// TIA Portal V17 export
// export: Created 2022-04-06T07:28:38.3800124Z, ExportSetting WithDefaults, DisplayName Totally Integrated Automation Portal, DisplayVersion V17, DisplayName TIA Portal Openness, DisplayVersion V17, DisplayName TIA Portal Version Control Interface, DisplayVersion V17, DisplayName TIA Portal Test Suite Advanced, DisplayVersion V17, DisplayName SINAMICS Startdrive Advanced, DisplayVersion V17, DisplayName SINAMICS Startdrive G130, G150, S120, S150, SINAMICS MV, S210, DisplayVersion V17, DisplayName SINAMICS Startdrive G110M, G120, G120C, G120D, G120P, G115D, DisplayVersion V17, DisplayName STEP 7 Professional, DisplayVersion V17, DisplayName STEP 7 Safety, DisplayVersion V17, DisplayName WinCC Advanced / Unified PC, DisplayVersion V17
FUNCTION_BLOCK "Motion"   // FB2, FBD
{ S7_Optimized_Access := 'TRUE' }
VERSION : 0.1
// stored: AutoNumber true, IsIECCheckEnabled true, IsRetainMemResEnabled false, MemoryReserve 100, SetENOAutomatically false, UDAEnableTagReadback false
   VAR
      MC_POWER_Instance { S7_SetPoint := 'True'} : MC_POWER;
      MC_RESET_Instance { S7_SetPoint := 'True'} : MC_RESET;
      MC_HOME_Instance { S7_SetPoint := 'True'} : MC_HOME;
      MC_MOVEVELOCITY_Instance { S7_SetPoint := 'True'} : MC_MOVEVELOCITY;
      MC_HALT_Instance { S7_SetPoint := 'True'} : MC_HALT;
      MC_POWER_Instance_1 { S7_SetPoint := 'True'} : MC_POWER;
      MC_RESET_Instance_1 { S7_SetPoint := 'True'} : MC_RESET;
      MC_HOME_Instance_1 { S7_SetPoint := 'True'} : MC_HOME;
      MC_MOVEVELOCITY_Instance_1 { S7_SetPoint := 'True'} : MC_MOVEVELOCITY;
      MC_HALT_Instance_1 { S7_SetPoint := 'True'} : MC_HALT;
      instMC_MOVEVELOCITY_SlsActive { S7_SetPoint := 'True'} : MC_MOVEVELOCITY;
      statSlsPtrig { S7_SetPoint := 'True'} : Bool;
   END_VAR
   VAR_TEMP   // added for the SCL form of the ladder/FBD networks
      _w1 : Bool;
   END_VAR
BEGIN

REGION Network 1
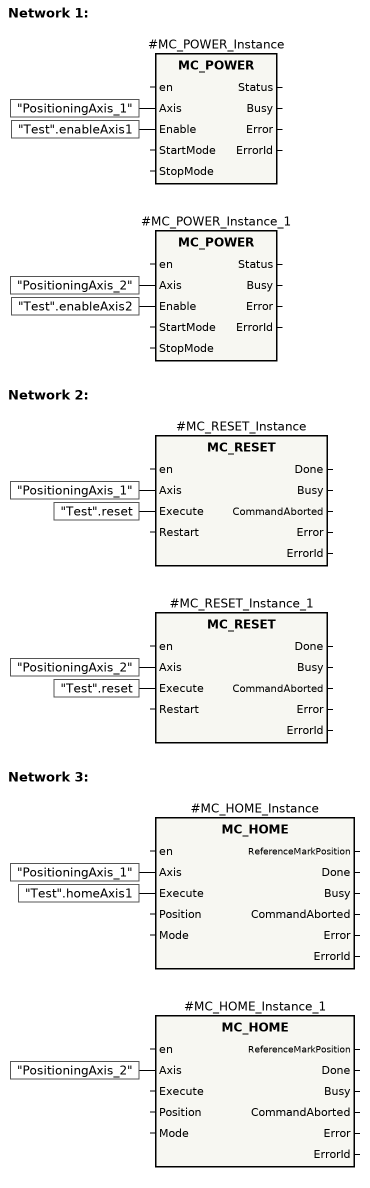
   #MC_POWER_Instance(Axis := "PositioningAxis_1", Enable := "Test".enableAxis1);   // MC_POWER
   #MC_POWER_Instance_1(Axis := "PositioningAxis_2", Enable := "Test".enableAxis2);   // MC_POWER
END_REGION

REGION Network 2
   #MC_RESET_Instance(Axis := "PositioningAxis_1", Execute := "Test".reset);   // MC_RESET
   #MC_RESET_Instance_1(Axis := "PositioningAxis_2", Execute := "Test".reset);   // MC_RESET
END_REGION

REGION Network 3
   #MC_HOME_Instance(Axis := "PositioningAxis_1", Execute := "Test".homeAxis1);   // MC_HOME
   #MC_HOME_Instance_1(Axis := "PositioningAxis_2");   // MC_HOME
END_REGION

REGION Network 4
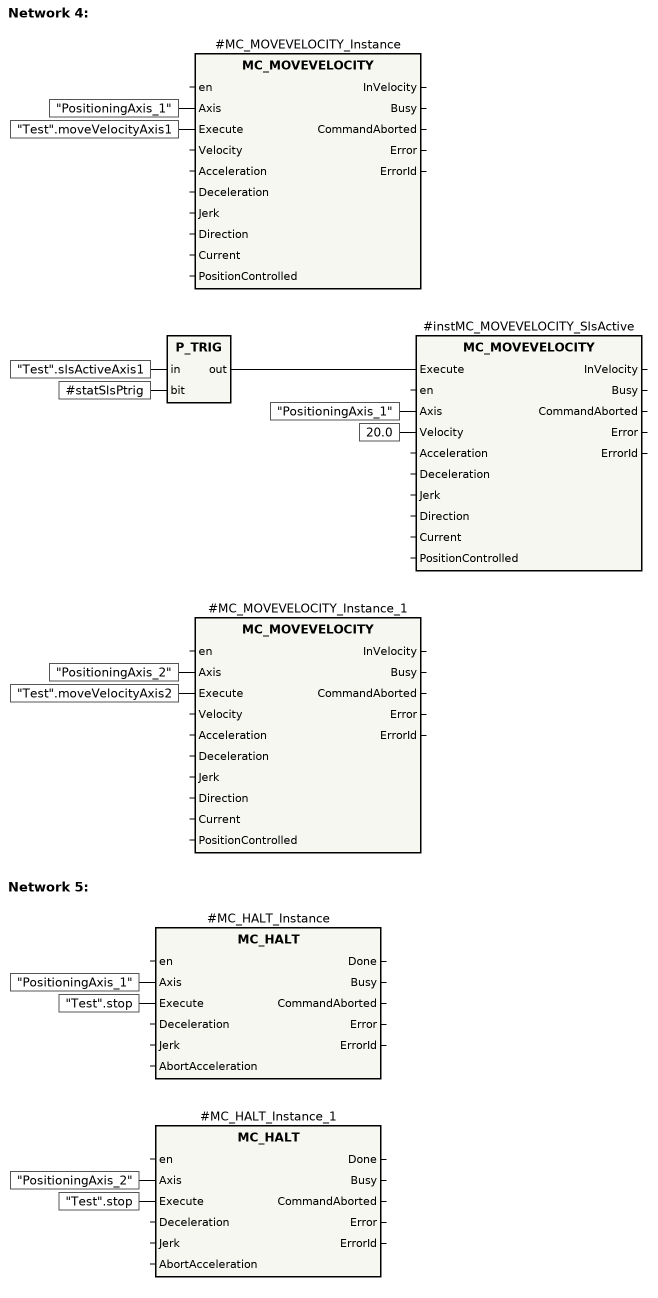
   #MC_MOVEVELOCITY_Instance(Axis := "PositioningAxis_1", Execute := "Test".moveVelocityAxis1);   // MC_MOVEVELOCITY
   #_w1 := "Test".slsActiveAxis1 AND NOT #statSlsPtrig;   // rising edge
   #statSlsPtrig := "Test".slsActiveAxis1;
   #instMC_MOVEVELOCITY_SlsActive(Execute := #_w1, Axis := "PositioningAxis_1", Velocity := 20.0);   // MC_MOVEVELOCITY
   #MC_MOVEVELOCITY_Instance_1(Axis := "PositioningAxis_2", Execute := "Test".moveVelocityAxis2);   // MC_MOVEVELOCITY
END_REGION

REGION Network 5
   #MC_HALT_Instance(Axis := "PositioningAxis_1", Execute := "Test".stop);   // MC_HALT
   #MC_HALT_Instance_1(Axis := "PositioningAxis_2", Execute := "Test".stop);   // MC_HALT
END_REGION
END_FUNCTION_BLOCK
